(*
SPDX-FileCopyrightText: © 2026 Oleksandr Tiutyk <trofimich@gmail.com>
SPDX-License-Identifier: MIT
License: https://opensource.org/license/mit
*)

(*!
<summary>Executes an ordered list of child activities one after another.</summary>
<description>
Advances at most one child activity per running step. When a child completes and a subsequent child exists,
the next child is selected as pending and started on the following running call. Suspending between two steps
pauses before the pending child starts; cancelling between steps completes cancellation without starting the
pending child. Resetting resets all non-ready child activities back to PASSIVE_READY and clears the selection.
</description>
*)

{attribute 'no_explicit_call' := 'do not call this function block directly'}
{attribute 'enable_dynamic_creation'}
FUNCTION_BLOCK SequenceActivity EXTENDS ExclusiveCompositeActivity
	IMPLEMENTS ISequenceActivity, TOF_Core.IConfigurationSerializable
VAR_STAT
	{attribute 'hide'}
	_ClassName : STRING := __POUNAME();
END_VAR
VAR
	{attribute 'OPC.UA.DA' := '0'}
	_Children : TOF_Collections.List<0>(valueValidator := 0);

	{attribute 'OPC.UA.DA' := '0'}
	_CurrentActivityIndex : DINT := Workflows.NO_SELECTED_ACTIVITY_INDEX;

	{attribute 'OPC.UA.DA' := '0'}
	_CurrentActivityStartPending : BOOL;
END_VAR

(*!
<summary>Appends a child activity to the sequence and assigns this sequence as its ParentActivity.</summary>
<description>
Requires PASSIVE_READY. Rejects null, self/ancestor cycles and children already attached elsewhere.
The child must be unattached, including to this parent; duplicate slots are rejected before insertion.
The parent chain and owning workflow must be PASSIVE_READY. Fixed workflow association is validated.
Storage allocation precedes parent callbacks; callback exceptions may leave a partial configuration.
Child references remain borrowed and must outlive the tree. No implicit detach or ownership transfer occurs.
</description>
<param name="activity">Child activity to append.</param>
*)
METHOD AddChildActivity
VAR_INPUT
	activity : IActivity;
END_VAR
VAR
	childParent : IWorkflowElement;
END_VAR
ValidateChildActivityAttachment(childActivity := activity, argumentName := 'activity');

childParent := activity.Parent;

IF childParent <> 0 THEN
	WorkflowExceptions.ThrowWorkflowAttachment(
		sourceNamespaceName := NamespaceName,
		sourceClassName := ClassName,
		sourcePOUName := __POUNAME(),
		sourcePosition := __POSITION(),
		message := "Child element already occupies a parent slot"
	);
END_IF

_Children.AppendGeneric(
	value := TOF_Core.GenericValueFactory.FromParts(
		genericTypeClass := TOF_Core.GENERIC_TYPE_CLASS.OBJECT,
		address := activity.SelfAddress,
		size := activity.SelfSize,
		memoryManagementBehavior := TOF_Core.GENERIC_MEMORY_MANAGEMENT_BEHAVIOR.STORE_ORIGINAL_REFERENCE_AND_NOT_OWNS_MEMORY
	)
);

activity.ParentActivity := THIS^;
END_METHOD

(*!
<summary>Borrows the initialized class name used in diagnostics.</summary>
<description>
Returns initialized metadata storage without allocation. Callers must not modify the returned string.
Derived function blocks must use distinct initialized static storage when overriding this metadata.
</description>
*)
{attribute 'monitoring' := 'call'}
PROPERTY ClassName : REFERENCE TO STRING
GET
ClassName REF= _ClassName;
END_GET
END_PROPERTY

(*!
<summary>Returns the child activity at CurrentActivityIndex, or 0 when no step is selected.</summary>
*)
{attribute 'monitoring' := 'call'}
PROPERTY FINAL CurrentActivity : IActivity
GET
IF _Children.Length > TOF_Core.SignedInt32.ZERO
	AND_THEN _CurrentActivityIndex >= TOF_Core.SignedInt32.ZERO
	AND_THEN _CurrentActivityIndex < _Children.Length
THEN
	__QUERYINTERFACE(_Children.Get(index := _CurrentActivityIndex).AsObject(), CurrentActivity);
END_IF
END_GET
END_PROPERTY

(*!
<summary>Returns the zero-based index of the currently selected child activity, or -1 when none is selected.</summary>
*)
{attribute 'monitoring' := 'call'}
PROPERTY FINAL CurrentActivityIndex : DINT
GET
CurrentActivityIndex := _CurrentActivityIndex;
END_GET
END_PROPERTY

(*!
<summary>Borrows the compiler-initialized library namespace.</summary>
<description>
Borrows storage from the live internal namespace provider. Reacquire references after application
reinitialization or relocation. Treat the reference as read-only; no ownership or synchronization is provided.
</description>
*)
{attribute 'monitoring' := 'call'}
PROPERTY NamespaceName : REFERENCE TO STRING
GET
NamespaceName REF= CurrentNamespace.Name;
END_GET
END_PROPERTY

(*!
<summary>Resets all non-ready child activities to PASSIVE_READY and clears the step selection.</summary>
<param name="startResetting">TRUE on the initial call from RequestReset.</param>
*)
METHOD PROTECTED OnResetting : ACTIVITY_RESETTING_STATE
VAR_INPUT
	startResetting : BOOL;
END_VAR
VAR
	i : DINT;
	childActivity : IActivity;
END_VAR
FOR i := 0 TO _Children.Length - 1 DO
	__QUERYINTERFACE(_Children.Get(index := i).AsObject(), childActivity);

	IF childActivity <> 0 AND_THEN childActivity.State <> WORKFLOW_ELEMENT_STATE.PASSIVE_READY THEN
		IF ResetChildActivity(childActivity := childActivity) = ACTIVITY_RESETTING_STATE.WORK_IN_PROGRESS THEN
			OnResetting := ACTIVITY_RESETTING_STATE.WORK_IN_PROGRESS;
			RETURN;
		END_IF
	END_IF
END_FOR

_CurrentActivityIndex := Workflows.NO_SELECTED_ACTIVITY_INDEX;
_CurrentActivityStartPending := FALSE;
OnResetting := ACTIVITY_RESETTING_STATE.WORK_RESET;
END_METHOD

(*!
<summary>Advances the current child activity by one step and selects the next child upon completion.</summary>
<param name="startRunning">TRUE on the initial call of a fresh start.</param>
<param name="startResuming">TRUE on the initial call when resuming from suspension.</param>
<param name="haltReason">Receives the child's HaltReason when the child halts.</param>
*)
METHOD PROTECTED OnRunning : ACTIVITY_RUNNING_STATE
VAR_INPUT
	startRunning : BOOL;
	startResuming : BOOL;
END_VAR
VAR_OUTPUT
	haltReason : WSTRING(255);
END_VAR
VAR
	activity : IActivity;
	
END_VAR
IF _Children.Length = TOF_Core.SignedInt32.ZERO THEN
	_CurrentActivityIndex := Workflows.NO_SELECTED_ACTIVITY_INDEX;
	_CurrentActivityStartPending := FALSE;
	OnRunning := ACTIVITY_RUNNING_STATE.WORK_COMPLETED;
	RETURN;
END_IF

IF startRunning OR_ELSE (startResuming AND_THEN _CurrentActivityIndex < TOF_Core.SignedInt32.ZERO) THEN
	_CurrentActivityIndex := TOF_Core.SignedInt32.ZERO;
	_CurrentActivityStartPending := TRUE;
END_IF

activity := CurrentActivity;

IF activity = 0 THEN
	TOF_Core.Exceptions.ThrowNullReference(
		sourceNamespaceName := NamespaceName,
		sourceClassName := ClassName,
		sourcePOUName := __POUNAME(),
		sourcePosition := __POSITION(),
		variableOrPropertyName := 'CurrentActivity'
	);
END_IF

IF startRunning OR_ELSE startResuming OR_ELSE _CurrentActivityStartPending THEN
	_CurrentActivityStartPending := FALSE;
	activity.RequestStart();
ELSE
	activity.Execute();
END_IF

OnRunning := MapChildRunningState(childState := activity.State);

IF OnRunning = ACTIVITY_RUNNING_STATE.WORK_HALTED THEN
	haltReason := activity.HaltReason;
ELSIF OnRunning = ACTIVITY_RUNNING_STATE.WORK_COMPLETED THEN
	selectNextActivity();

	IF _CurrentActivityIndex >= TOF_Core.SignedInt32.ZERO THEN
		OnRunning := ACTIVITY_RUNNING_STATE.WORK_IN_PROGRESS;
	END_IF
END_IF
END_METHOD

(*!
<summary>Stops the active child activity or stops immediately at a pending step boundary.</summary>
<param name="startCancelling">TRUE on the initial call from RequestCancel.</param>
<param name="startSuspending">TRUE on the initial call from RequestSuspend.</param>
<param name="haltReason">Receives the child's HaltReason if the child halts while stopping.</param>
*)
METHOD PROTECTED OnStopping : ACTIVITY_STOPPING_STATE
VAR_INPUT
	startCancelling : BOOL;
	startSuspending : BOOL;
END_VAR
VAR_OUTPUT
	haltReason : WSTRING(255);
END_VAR
VAR
	activity : IActivity;
END_VAR
IF _Children.Length = TOF_Core.SignedInt32.ZERO THEN
	OnStopping := ACTIVITY_STOPPING_STATE.WORK_COMPLETED;
	RETURN;
END_IF

activity := CurrentActivity;

IF activity = 0 THEN
	IF startCancelling OR_ELSE startSuspending THEN
		OnStopping := ACTIVITY_STOPPING_STATE.WORK_STOPPED;
	ELSE
		OnStopping := ACTIVITY_STOPPING_STATE.WORK_COMPLETED;
	END_IF

	RETURN;
END_IF

IF _CurrentActivityStartPending THEN
	OnStopping := ACTIVITY_STOPPING_STATE.WORK_STOPPED;
	RETURN;
END_IF

IF NOT activity.Busy THEN
	IF startCancelling AND_THEN activity.State = WORKFLOW_ELEMENT_STATE.PASSIVE_SUSPENDED THEN
		activity.RequestCancel(reason := _CancelReason);
	END_IF

	OnStopping := MapChildStoppingState(childState := activity.State);

	IF OnStopping = ACTIVITY_STOPPING_STATE.WORK_HALTED THEN
		haltReason := activity.HaltReason;
	END_IF

	RETURN;
END_IF

IF startCancelling THEN
	activity.RequestCancel(reason := _CancelReason);
ELSIF startSuspending THEN
	activity.RequestSuspend();
ELSE
	activity.Execute();
END_IF

OnStopping := MapChildStoppingState(childState := activity.State);

IF OnStopping = ACTIVITY_STOPPING_STATE.WORK_HALTED THEN
	haltReason := activity.HaltReason;
END_IF
END_METHOD

(*!
<summary>Selects the next child activity in sequence as pending, or clears the selection after the last child.</summary>
*)
METHOD PRIVATE selectNextActivity
IF _CurrentActivityIndex < _Children.Length - 1 THEN
	_CurrentActivityIndex := _CurrentActivityIndex + 1;
	_CurrentActivityStartPending := TRUE;
ELSE
	_CurrentActivityIndex := Workflows.NO_SELECTED_ACTIVITY_INDEX;
	_CurrentActivityStartPending := FALSE;
END_IF
END_METHOD

(*!
<summary>Reports the size of this concrete function block instance in bytes.</summary>
<description>
Reports the instance layout rather than dynamic allocations owned by its fields. A derived function block
with a different layout must override this property; the value does not grant disposal rights.
</description>
*)
{attribute 'monitoring' := 'call'}
PROPERTY SelfSize : ULINT
GET
SelfSize := XSIZEOF(THIS^);
END_GET
END_PROPERTY

(*!
<summary>Writes the configuration fields for this object.</summary>
<description>Borrows the writer for this call. A failure invalidates the current output document.</description>
*)
METHOD Serialize
VAR_INPUT
	writer : TOF_Core.IConfigurationWriter;
END_VAR
VAR
	i : DINT;
END_VAR
Workflows.WriteConfigurationHeader(writer := writer, source := THIS^, displayName := Name, scope := THIS^);
writer.BeginArray(name := 'children');

FOR i := 0 TO _Children.Length - 1 DO
	Workflows.WriteConfigurationObject(writer := writer, name := '', source := _Children.Get(index := i).AsObject());
END_FOR

writer.EndArray();
END_METHOD

(*!
<summary>Restores this fresh instance from its configuration object.</summary>
<description>
The reader, document node and deserialization context are borrowed for this call.
On failure discard the partial instance.
</description>
<param name="reader">Active configuration reader.</param>
<param name="node">Configuration node for this activity.</param>
<param name="context">Active configuration deserialization context providing workflow reconstruction services.</param>
*)
METHOD Deserialize
VAR_INPUT
	reader : TOF_Core.IConfigurationReader;
	node : TOF_Core.CONFIGURATION_NODE;
	context : TOF_Core.IConfigurationDeserializationContext;
END_VAR
VAR
	loader : IWorkflowLoader;
	items : TOF_Core.CONFIGURATION_NODE;
	count : DINT;
	i : DINT;
END_VAR
loader := WorkflowConfigurationSerializer.ResolveWorkflowLoader(context := context);
Workflows.ReadConfigurationHeader(reader := reader, node := node, target := THIS^, scope := THIS^);

items := reader.GetField(node := node, name := 'children');
count := TO_DINT(reader.GetArraySize(node := items));

FOR i := 0 TO count - 1 DO
	AddChildActivity(
		activity := Workflows.ReadActivity(loader := loader, node := reader.GetItem(node := items, index := TO_UDINT(i)))
	);
END_FOR
END_METHOD

END_FUNCTION_BLOCK

(* stored: Version 1.1.0.1
   POU SequenceActivity: Id {1bca36af-b7de-4b08-b287-296cf8c67b1e}, SpecialFunc None
   Folder Overriden methods: Id {c5874289-fa30-4e42-9a18-d42194d8091a}
   Folder Service methods: Id {3f51cbe1-be68-4e5e-a663-f6baed6e006e}
   Method AddChildActivity: Id {a30975d8-8e95-48ec-a5ab-8e9aa1d75be7}
   Property ClassName: Id {72010df4-c4eb-4a27-acd3-c42588cae27a}
   Get Get: Id {d41e15da-8455-40c4-82b6-9574b0fe558a}
   Property CurrentActivity: Id {1a4ebfb1-244f-44f9-8b12-8787ad4a03a7}
   Get Get: Id {3a9f72bd-ef17-4fe7-b05f-5afb314fb2fe}
   Property CurrentActivityIndex: Id {8fdd1d3f-3fdc-492f-b895-9e1e6061e1cd}
   Get Get: Id {1ac1fa84-8eed-4de1-9a51-3f86182c90ee}
   Property NamespaceName: Id {1771b04b-38be-4416-9a7e-972d57af0862}
   Get Get: Id {d41be4b9-0e62-4695-98dc-b4b063425079}
   Method OnResetting: Id {7b20c640-7f05-4729-b6d4-37b7999c102f}
   Method OnRunning: Id {53e0829c-4dbd-4b85-a474-dd611d0f45cd}
   Method OnStopping: Id {58c42973-4e56-4492-9a0d-c7eb58c052dc}
   Method selectNextActivity: Id {7ad99828-ec1f-4f8b-bfdb-f4b31de1f87c}
   Property SelfSize: Id {41f1ba7d-873e-4cab-8142-5d65c440edef}
   Get Get: Id {3d49e29e-d473-48e0-b330-20e133f0a344}
   Method Serialize: Id {57353df2-319f-4bca-938b-1f6be3fec8a9}
   Method Deserialize: Id {5fb419d4-4e58-45d9-ae31-84af188e24f4} *)
